# EPICS autosave request: iocs/axisSXR40IOC/iocBoot/iocAxisSXR40/auto_settings.req
# Settings restored on IOC restart, saved every 30 s by the create_monitor_set
# call at the end of st.cmd.
#
# axisSXR40_settings.req is found via set_requestfile_path("$(ADAXISSXR40)/axisSXR40App/Db");
# the NDStdArrays and commonPlugin request files come from the paths
# commonPlugins.cmd adds ($(ADCORE)/db and $(ADCORE)/iocBoot).
#
# axisSXR40_settings.req still lists the 8 parameters this camera does not
# implement (auto-exposure, CMS/HDR image mode, defect correction, enhance, black
# level, brightness, sharpness, HDR-K). save_restore logs those as missing PVs
# rather than failing -- see Known gaps in README.md.

file "axisSXR40_settings.req",     P=$(P),  R=cam1:
file "NDStdArrays_settings.req",   P=$(P),  R=image1:
file "commonPlugin_settings.req",  P=$(P)
